{attribute addProperty BoxType "EL2602-0010-0016"}
{attribute addProperty Id "InputsAT %I*Inputs_BDF19946810ChannelAT %Q*ARRAY[0..1] OF Channel_7F374EB01620WcStateAT %I*WcState_F855686C1620InfoDataAT %I*InfoData_192954DE1620"}
{attribute addProperty CRC "772639126"}
{attribute addProperty SizeInBites "56"}
{attribute addProperty SizeInBytes "7"}
TYPE EL2602_0939F1F7 :
STRUCT
	{attribute addProperty Name "Inputs"}
	Inputs : Inputs_BDF19946;
	{attribute addProperty Name "Channel"}
	Channel : ARRAY[0..1] OF Channel_7F374EB0;
	{attribute addProperty Name "WcState"}
	WcState : WcState_F855686C;
	{attribute addProperty Name "InfoData"}
	InfoData : InfoData_192954DE;
END_STRUCT
END_TYPE

(* stored: Version 1.2.0.0, ProductVersion 3.1.4024.9
   DUT EL2602_0939F1F7: Id {d873d290-e0e9-41c5-9aec-8f51436bf72f} *)
